FUNCTION IsLessThanOrEqualAnyType : BOOL
VAR_INPUT
	a					: __SYSTEM.AnyType; // A and B have to be same type
	b					: __SYSTEM.AnyType; // A and B have to be same type
END_VAR

IsLessThanOrEqualAnyType := NOT IsGreaterThanAnyType(a, b);

END_FUNCTION

(* stored: Version 1.1.0.1
   POU IsLessThanOrEqualAnyType: Id {2b1c8f92-0781-0e7b-2091-b8bea93306d5}, SpecialFunc None *)
